Fanuc KAREL source: kt00754.KL

-- PROVISIONAL review KL for V1013-1; original PC SHA256 de0b9bebfac8fffbbe1da65d0391fbd0fcb3d93cd2c8558811e3e084cb03ae9e
-- Incomplete behavior may be omitted. Consult companion uncertainty JSON. Do not deploy.
PROGRAM KT00754
%NOLOCKGROUP
VAR
  OUT : INTEGER
-- UNRESOLVED_DECL H1 type=002017
-- UNRESOLVED_DECL H2 type=002017
BEGIN
  -- UNRESOLVED_PC offsets 5-19; opcodes 2E,22,9D,33,B4
  -- UNRESOLVED_PC offsets 24-38; opcodes 2E,22,9D,33,B4
  -- UNRESOLVED_PC offsets 43-57; opcodes 2E,22,9D,33,B4
  -- UNRESOLVED_PC offsets 62-76; opcodes 2E,22,9D,33,B4
  -- UNRESOLVED_PC offsets 81-97; opcodes 22,9D,33,B3,50,23
  -- UNRESOLVED_PC offsets 102-106; opcodes 7F
END KT00754
